// TIA Portal V18 program export: 1 tag tables, 0 data types, 0 data blocks, 2 code blocks (in call order from the OBs), 1 instance data blocks

VAR_GLOBAL   // PLC tag table "AI_PLC_Tags_CIP_Mixing"
   AI_LT3203_PV AT %MD200 : Real;   // Mức bồn trộn 1 LT3203 (0.0 đến 1000.0 L)
   AI_TT3204_PV AT %MD204 : Real;   // Nhiệt độ bồn trộn 1 TT3204 (0.0 đến 100.0 °C)
   AI_LT3209_PV AT %MD208 : Real;   // Mức bồn trộn 2 LT3209 (0.0 đến 1000.0 L)
   AI_TT3208_PV AT %MD212 : Real;   // Nhiệt độ bồn trộn 2 TT3208 (0.0 đến 100.0 °C)
   AI_LT3213_PV AT %MD216 : Real;   // Mức bồn trộn 3 LT3213 (0.0 đến 1000.0 L)
   AI_TT3214_PV AT %MD220 : Real;   // Nhiệt độ bồn trộn 3 TT3214 (0.0 đến 100.0 °C)
   AI_LT3218_PV AT %MD224 : Real;   // Mức bồn trộn 4 LT3218 (0.0 đến 1000.0 L)
   AI_TT3219_PV AT %MD228 : Real;   // Nhiệt độ bồn trộn 4 TT3219 (0.0 đến 100.0 °C)
   AI_BON1_Chay AT %M232.0 : Bool;   // Báo trạng thái bồn trộn 1 đang chạy
   AI_BON2_Chay AT %M232.1 : Bool;   // Báo trạng thái bồn trộn 2 đang chạy
   AI_BON3_Chay AT %M232.2 : Bool;   // Báo trạng thái bồn trộn 3 đang chạy
   AI_BON4_Chay AT %M232.3 : Bool;   // Báo trạng thái bồn trộn 4 đang chạy
   AI_PUMP3264_Chay AT %M232.4 : Bool;   // Trạng thái chạy của bơm PUMP3264
   AI_PUMP3265_Chay AT %M232.5 : Bool;   // Trạng thái chạy của bơm PUMP3265
   AI_Logged_In AT %MW234 : Int;   // Trạng thái đăng nhập trên HMI
   Sim_Counter AT %MD236 : Real;   // Biến đếm trung gian cho sóng tam giác mô phỏng
   Sim_Dir AT %M240.0 : Bool;   // Bit hướng đếm mô phỏng (0: Tăng, 1: Giảm)
   Sim_Val_Norm AT %MD242 : Real;   // Giá trị đếm đã chuẩn hóa về dải 0.0 - 1.0
   Timer_Sim_Pulse_Output AT %M240.1 : Bool;   // Xung kích hoạt đếm từ Timer
END_VAR

ORGANIZATION_BLOCK "Main"   // OB1, LAD, ProgramCycle
{ S7_Optimized_Access := 'TRUE' }
VERSION : 0.1
// stored: AutoNumber true, IsIECCheckEnabled false
   VAR_INPUT
      Initial_Call : Bool;
      Remanence : Bool;
   END_VAR
BEGIN

REGION Network 1: Gọi khối mô phỏng cảm biến SCADA
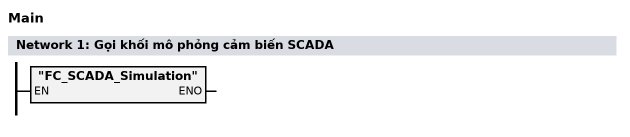
   RUNG wire#powerrail
      "FC_SCADA_Simulation"()
   END_RUNG
   // the same network as SCL:
   "FC_SCADA_Simulation"();
END_REGION
END_ORGANIZATION_BLOCK

FUNCTION "FC_SCADA_Simulation" : Void   // FC10, LAD
{ S7_Optimized_Access := 'TRUE' }
VERSION : 0.1
// stored: AutoNumber true, IsIECCheckEnabled false
BEGIN

REGION Network 1: Tạo xung kích hoạt chu kỳ mô phỏng (50ms)
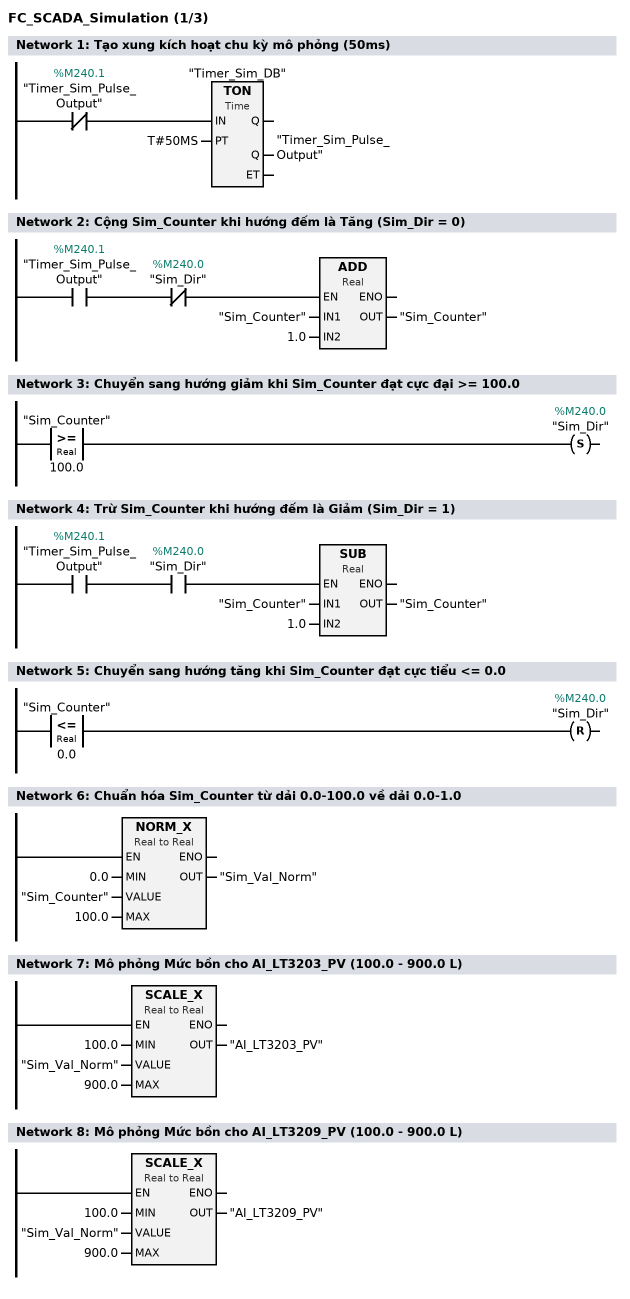
   RUNG wire#powerrail
      I_Contact( "Timer_Sim_Pulse_Output" )
      { S7_Templates := "time_type := Time" } "Timer_Sim_DB".TON(pt := T#50MS, q => "Timer_Sim_Pulse_Output", et =>)
   END_RUNG
   // the same network as SCL:
   "Timer_Sim_DB".TON(IN := NOT "Timer_Sim_Pulse_Output", PT := T#50MS, Q => "Timer_Sim_Pulse_Output");
END_REGION

REGION Network 2: Cộng Sim_Counter khi hướng đếm là Tăng (Sim_Dir = 0)
   RUNG wire#powerrail
      Contact( "Timer_Sim_Pulse_Output" )
      I_Contact( "Sim_Dir" )
      { S7_Templates := "SrcType := Real"; S7_GenerateENO := "TRUE" } Add(in1 := "Sim_Counter", in2 := 1.0, out => "Sim_Counter")
   END_RUNG
   // the same network as SCL:
   IF "Timer_Sim_Pulse_Output" AND NOT "Sim_Dir" THEN "Sim_Counter" := "Sim_Counter" + 1.0; END_IF;
END_REGION

REGION Network 3: Chuyển sang hướng giảm khi Sim_Counter đạt cực đại >= 100.0
   RUNG wire#powerrail
      { S7_Templates := "SrcType := Real" } GE_Contact(in1 := "Sim_Counter", in2 := 100.0)
      S_Coil( "Sim_Dir" )
   END_RUNG
   // the same network as SCL:
   IF "Sim_Counter" >= 100.0 THEN "Sim_Dir" := TRUE; END_IF;
END_REGION

REGION Network 4: Trừ Sim_Counter khi hướng đếm là Giảm (Sim_Dir = 1)
   RUNG wire#powerrail
      Contact( "Timer_Sim_Pulse_Output" )
      Contact( "Sim_Dir" )
      { S7_Templates := "SrcType := Real"; S7_GenerateENO := "TRUE" } Sub(in1 := "Sim_Counter", in2 := 1.0, out => "Sim_Counter")
   END_RUNG
   // the same network as SCL:
   IF "Timer_Sim_Pulse_Output" AND "Sim_Dir" THEN "Sim_Counter" := "Sim_Counter" - 1.0; END_IF;
END_REGION

REGION Network 5: Chuyển sang hướng tăng khi Sim_Counter đạt cực tiểu <= 0.0
   RUNG wire#powerrail
      { S7_Templates := "SrcType := Real" } LE_Contact(in1 := "Sim_Counter", in2 := 0.0)
      R_Coil( "Sim_Dir" )
   END_RUNG
   // the same network as SCL:
   IF "Sim_Counter" <= 0.0 THEN "Sim_Dir" := FALSE; END_IF;
END_REGION

REGION Network 6: Chuẩn hóa Sim_Counter từ dải 0.0-100.0 về dải 0.0-1.0
   RUNG wire#powerrail
      { S7_Templates := "[SrcType := Real, DestType := Real]" } Normalize(min := 0.0, value := "Sim_Counter", max := 100.0, out => "Sim_Val_Norm")
   END_RUNG
   // the same network as SCL:
   "Sim_Val_Norm" := NORM_X(MIN := 0.0, VALUE := "Sim_Counter", MAX := 100.0);
END_REGION

REGION Network 7: Mô phỏng Mức bồn cho AI_LT3203_PV (100.0 - 900.0 L)
   RUNG wire#powerrail
      { S7_Templates := "[SrcType := Real, DestType := Real]" } Scale(min := 100.0, value := "Sim_Val_Norm", max := 900.0, out => "AI_LT3203_PV")
   END_RUNG
   // the same network as SCL:
   "AI_LT3203_PV" := SCALE_X(MIN := 100.0, VALUE := "Sim_Val_Norm", MAX := 900.0);
END_REGION

REGION Network 8: Mô phỏng Mức bồn cho AI_LT3209_PV (100.0 - 900.0 L)
   RUNG wire#powerrail
      { S7_Templates := "[SrcType := Real, DestType := Real]" } Scale(min := 100.0, value := "Sim_Val_Norm", max := 900.0, out => "AI_LT3209_PV")
   END_RUNG
   // the same network as SCL:
   "AI_LT3209_PV" := SCALE_X(MIN := 100.0, VALUE := "Sim_Val_Norm", MAX := 900.0);
END_REGION

REGION Network 9: Mô phỏng Mức bồn cho AI_LT3213_PV (100.0 - 900.0 L)
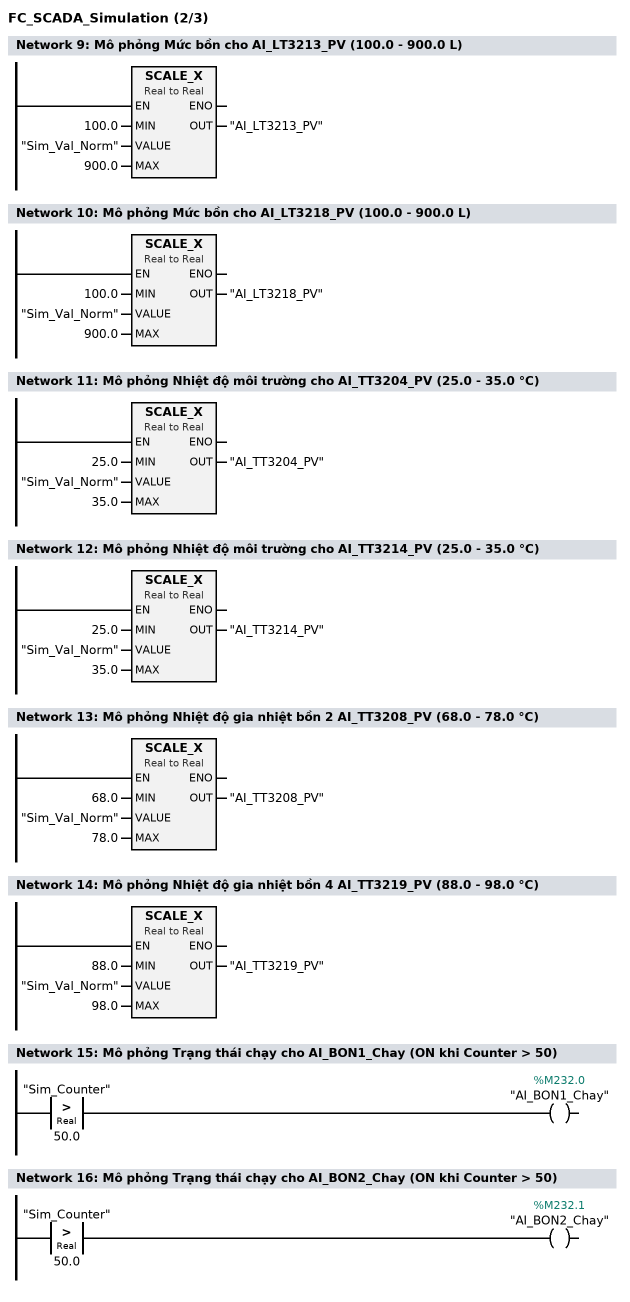
   RUNG wire#powerrail
      { S7_Templates := "[SrcType := Real, DestType := Real]" } Scale(min := 100.0, value := "Sim_Val_Norm", max := 900.0, out => "AI_LT3213_PV")
   END_RUNG
   // the same network as SCL:
   "AI_LT3213_PV" := SCALE_X(MIN := 100.0, VALUE := "Sim_Val_Norm", MAX := 900.0);
END_REGION

REGION Network 10: Mô phỏng Mức bồn cho AI_LT3218_PV (100.0 - 900.0 L)
   RUNG wire#powerrail
      { S7_Templates := "[SrcType := Real, DestType := Real]" } Scale(min := 100.0, value := "Sim_Val_Norm", max := 900.0, out => "AI_LT3218_PV")
   END_RUNG
   // the same network as SCL:
   "AI_LT3218_PV" := SCALE_X(MIN := 100.0, VALUE := "Sim_Val_Norm", MAX := 900.0);
END_REGION

REGION Network 11: Mô phỏng Nhiệt độ môi trường cho AI_TT3204_PV (25.0 - 35.0 °C)
   RUNG wire#powerrail
      { S7_Templates := "[SrcType := Real, DestType := Real]" } Scale(min := 25.0, value := "Sim_Val_Norm", max := 35.0, out => "AI_TT3204_PV")
   END_RUNG
   // the same network as SCL:
   "AI_TT3204_PV" := SCALE_X(MIN := 25.0, VALUE := "Sim_Val_Norm", MAX := 35.0);
END_REGION

REGION Network 12: Mô phỏng Nhiệt độ môi trường cho AI_TT3214_PV (25.0 - 35.0 °C)
   RUNG wire#powerrail
      { S7_Templates := "[SrcType := Real, DestType := Real]" } Scale(min := 25.0, value := "Sim_Val_Norm", max := 35.0, out => "AI_TT3214_PV")
   END_RUNG
   // the same network as SCL:
   "AI_TT3214_PV" := SCALE_X(MIN := 25.0, VALUE := "Sim_Val_Norm", MAX := 35.0);
END_REGION

REGION Network 13: Mô phỏng Nhiệt độ gia nhiệt bồn 2 AI_TT3208_PV (68.0 - 78.0 °C)
   RUNG wire#powerrail
      { S7_Templates := "[SrcType := Real, DestType := Real]" } Scale(min := 68.0, value := "Sim_Val_Norm", max := 78.0, out => "AI_TT3208_PV")
   END_RUNG
   // the same network as SCL:
   "AI_TT3208_PV" := SCALE_X(MIN := 68.0, VALUE := "Sim_Val_Norm", MAX := 78.0);
END_REGION

REGION Network 14: Mô phỏng Nhiệt độ gia nhiệt bồn 4 AI_TT3219_PV (88.0 - 98.0 °C)
   RUNG wire#powerrail
      { S7_Templates := "[SrcType := Real, DestType := Real]" } Scale(min := 88.0, value := "Sim_Val_Norm", max := 98.0, out => "AI_TT3219_PV")
   END_RUNG
   // the same network as SCL:
   "AI_TT3219_PV" := SCALE_X(MIN := 88.0, VALUE := "Sim_Val_Norm", MAX := 98.0);
END_REGION

REGION Network 15: Mô phỏng Trạng thái chạy cho AI_BON1_Chay (ON khi Counter > 50)
   RUNG wire#powerrail
      { S7_Templates := "SrcType := Real" } GT_Contact(in1 := "Sim_Counter", in2 := 50.0)
      Coil( "AI_BON1_Chay" )
   END_RUNG
   // the same network as SCL:
   "AI_BON1_Chay" := "Sim_Counter" > 50.0;
END_REGION

REGION Network 16: Mô phỏng Trạng thái chạy cho AI_BON2_Chay (ON khi Counter > 50)
   RUNG wire#powerrail
      { S7_Templates := "SrcType := Real" } GT_Contact(in1 := "Sim_Counter", in2 := 50.0)
      Coil( "AI_BON2_Chay" )
   END_RUNG
   // the same network as SCL:
   "AI_BON2_Chay" := "Sim_Counter" > 50.0;
END_REGION

REGION Network 17: Mô phỏng Trạng thái chạy cho AI_BON3_Chay (ON khi Counter > 50)
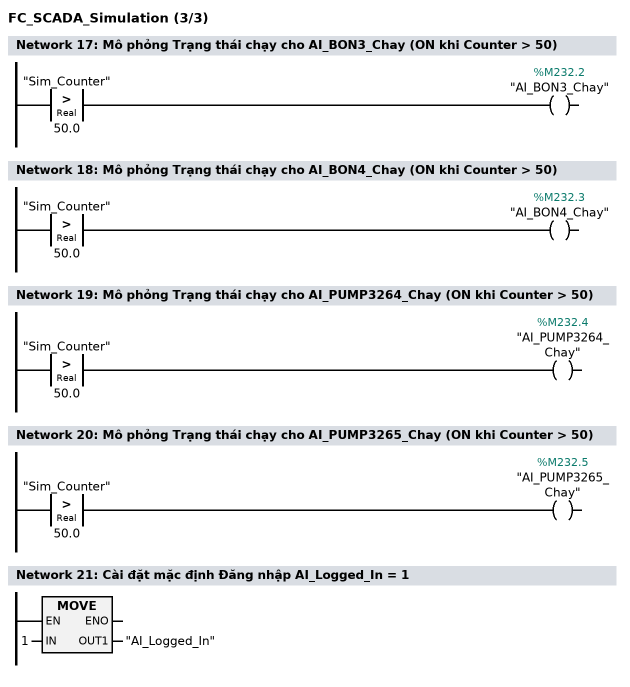
   RUNG wire#powerrail
      { S7_Templates := "SrcType := Real" } GT_Contact(in1 := "Sim_Counter", in2 := 50.0)
      Coil( "AI_BON3_Chay" )
   END_RUNG
   // the same network as SCL:
   "AI_BON3_Chay" := "Sim_Counter" > 50.0;
END_REGION

REGION Network 18: Mô phỏng Trạng thái chạy cho AI_BON4_Chay (ON khi Counter > 50)
   RUNG wire#powerrail
      { S7_Templates := "SrcType := Real" } GT_Contact(in1 := "Sim_Counter", in2 := 50.0)
      Coil( "AI_BON4_Chay" )
   END_RUNG
   // the same network as SCL:
   "AI_BON4_Chay" := "Sim_Counter" > 50.0;
END_REGION

REGION Network 19: Mô phỏng Trạng thái chạy cho AI_PUMP3264_Chay (ON khi Counter > 50)
   RUNG wire#powerrail
      { S7_Templates := "SrcType := Real" } GT_Contact(in1 := "Sim_Counter", in2 := 50.0)
      Coil( "AI_PUMP3264_Chay" )
   END_RUNG
   // the same network as SCL:
   "AI_PUMP3264_Chay" := "Sim_Counter" > 50.0;
END_REGION

REGION Network 20: Mô phỏng Trạng thái chạy cho AI_PUMP3265_Chay (ON khi Counter > 50)
   RUNG wire#powerrail
      { S7_Templates := "SrcType := Real" } GT_Contact(in1 := "Sim_Counter", in2 := 50.0)
      Coil( "AI_PUMP3265_Chay" )
   END_RUNG
   // the same network as SCL:
   "AI_PUMP3265_Chay" := "Sim_Counter" > 50.0;
END_REGION

REGION Network 21: Cài đặt mặc định Đăng nhập AI_Logged_In = 1
   RUNG wire#powerrail
      { S7_GenerateENO := "TRUE" } Move(in := 1, out1 => "AI_Logged_In")
   END_RUNG
   // the same network as SCL:
   "AI_Logged_In" := 1;
END_REGION
END_FUNCTION

DATA_BLOCK "Timer_Sim_DB"   // DB10
TITLE = Timer_Sim_DB
// DB chứa biến đếm thời gian cho khối mô phỏng
// stored: AutoNumber true, InstanceOfName IEC_TIMER, OfSystemLibElement IEC_TIMER, OfSystemLibVersion 1.0
"IEC_TIMER"
   // VAR
   //    PT : Time;
   //    ET { ExternalWritable := 'False'} : Time;
   //    IN : Bool;
   //    Q { ExternalWritable := 'False'} : Bool;
   // END_VAR
BEGIN
END_DATA_BLOCK
